Yaskawa INFORM job: FMTV_BACK_HOME.JBI

/JOB
//NAME FMTV_BACK_HOME
//POS
///NPOS 4,0,0,0,0,0
///TOOL 0
///POSTYPE PULSE
///PULSE
C00000=-47368,-58389,-75463,-75325,82045,-91552
C00001=-47368,-166672,-122912,-75325,82045,-91552
C00002=-47368,-169255,14547,-75325,114153,-156925
C00003=-63952,-155163,126853,-105316,-81596,-126671
//INST
///DATE 2022/03/21 15:43
///ATTR SC,RW
///GROUP1 RB1
NOP
MOVJ C00000 VJ=65.00  //BIT CHANGE
MOVJ C00001 VJ=65.00
MOVJ C00002 VJ=65.00
MOVJ C00003 VJ=65.00  //HOME
END
